// TIA Portal V16 export
// export: Created 2020-03-07T16:06:13.7080048Z, ExportSetting WithDefaults, DisplayName Totally Integrated Automation Portal, DisplayVersion V16 Update 1, DisplayName TIA Portal Version Control Interface, DisplayVersion V16, DisplayName TIA Portal Openness, DisplayVersion V16 Update 1, DisplayName STEP 7 Professional, DisplayVersion V16 Update 1, DisplayName STEP 7 Safety, DisplayVersion V16, DisplayName WinCC Professional, DisplayVersion V16 Update 1
FUNCTION "function" : Void   // FC1, LAD
{ S7_Optimized_Access := 'TRUE' }
VERSION : 0.1
// stored: AutoNumber true, IsIECCheckEnabled false, SetENOAutomatically false, UDAEnableTagReadback false
   VAR_INPUT
      abc : Bool;
   END_VAR
   VAR_OUTPUT
      output : Bool;
   END_VAR
   VAR_TEMP
      intermediate : Bool;
   END_VAR
   VAR_TEMP   // added for the SCL form of the ladder/FBD networks
      _w1 : Bool;
   END_VAR
BEGIN

REGION Network 1
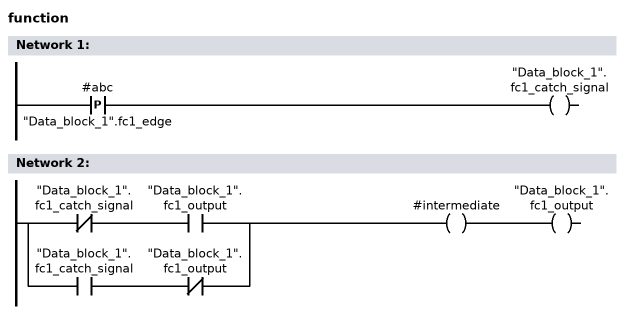
   RUNG wire#powerrail
      P_Contact(operand := #abc, bit := "Data_block_1".fc1_edge)
      Coil( "Data_block_1".fc1_catch_signal )
   END_RUNG
   // the same network as SCL:
   #_w1 := #abc AND NOT "Data_block_1".fc1_edge;   // rising edge of #abc
   "Data_block_1".fc1_edge := #abc;
   "Data_block_1".fc1_catch_signal := #_w1;
END_REGION

REGION Network 2
   RUNG wire#powerrail
      I_Contact( "Data_block_1".fc1_catch_signal )
      Contact( "Data_block_1".fc1_output )
      wire#w1
      Coil( #intermediate )
      Coil( "Data_block_1".fc1_output )
   END_RUNG
   RUNG wire#powerrail
      Contact( "Data_block_1".fc1_catch_signal )
      I_Contact( "Data_block_1".fc1_output )
   END_RUNG wire#w1
   // the same network as SCL:
   #intermediate := (NOT "Data_block_1".fc1_catch_signal AND "Data_block_1".fc1_output) OR ("Data_block_1".fc1_catch_signal AND NOT "Data_block_1".fc1_output);
   "Data_block_1".fc1_output := #intermediate;
END_REGION
END_FUNCTION
